ABB RobotStudio station: proyecto1.2.rsstn

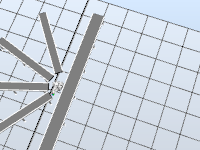
Station proyecto1.2 (saved by RobotStudio 20.4.9280.0)
Layout (positions relative to the parent item):
  - IRB140_6_81_C_03 [mechanism, from Robots\IRB140_6_81_C_G_03.rslib] at (4211.58, -254.35, 0) mm, rotated rx 0 ry 0 rz 179.86 deg; joint values [0, 0, 0, 0, 0.5236, 0] (rad or m)
  - Banda_cajas [part] at (0, -1120.44, 0) mm
  - IRB140_6_81_C_03_2 [mechanism, from Robots\IRB140_6_81_C_G_03.rslib] at (-657.92, -762.72, 0) mm; joint values [0, 0, 0, 0, 0.5236, 0] (rad or m)
  - EPAL 6 half pallet [part] at (-887.28, -1772.67, 0) mm
  - Banda_Psopa [part] at (4862.11, -266.95, 0) mm, rotated rx 0 ry 0 rz -54 deg
  - Banda_PSeco [part] at (4556.38, 48.6, 0) mm, rotated rx 0 ry 0 rz -18 deg
  - Banda_PPostre [part] at (3738.83, 27.98, 0) mm, rotated rx 0 ry 0 rz 54 deg
  - Banda_Posillo [part] at (4146.52, 149.17, 0) mm, rotated rx 0 ry 0 rz 18 deg
